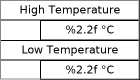
VISUALIZATION UI_Temp  // 140x80
VAR_IN_OUT
	setting		: Room_Settings_TemperatureSettings;
END_VAR
    Rectangle (0,40 140x20), "Low Temperature"
    Rectangle (40,60 100x20), "%2.2f °C", text variable: setting.rLow
        OnMouseClick: write the text variable via Default
    Rectangle (0,0 140x20), "High Temperature"
    Rectangle (40,20 100x20), "%2.2f °C", text variable: setting.rHigh
        OnMouseClick: write the text variable via Default
END_VISUALIZATION

(* stored: Version 1.1.0.1
   Visu UI_Temp: Id {2379e8c6-56b5-44b9-8913-a70060ae4e23} *)
